// TIA Portal V20 export
VAR_GLOBAL   // PLC tag table "Default tag table"
   SAFETY_TEST AT %M200.0 : Bool;
   Tag_1 AT %M200.1 : Bool;
   Tag_3 AT %M2000.0 : Bool;
   Tag_4 AT %M2000.1 : Bool;
   armsMainValve AT %Q1557.0 : Bool;
   clampsMainValve AT %Q1557.1 : Bool;
   Tag_5 AT %M2001.0 : Bool;
   Tag_6 AT %M2001.1 : Bool;
   Tag_7 AT %M2001.3 : Bool;
   Tag_8 AT %M2001.2 : Bool;
   Tag_9 AT %M222.2 : Bool;
   SS2_R1_STO AT %Q150.0 : Bool;
   Tag_11 AT %M222.3 : Bool;
   Tag_10 AT %M212.0 : Bool;
   Tag_12 AT %M500.0 : Bool;
   Tag_13 AT %M500.1 : Bool;
   Tag_14 AT %M500.2 : Bool;
   Tag_15 AT %M501.0 : Bool;
   Tag_16 AT %M501.1 : Bool;
   TipHydContactorFB AT %I2105.0 : Bool;
   S2_R2_STO AT %Q169.0 : Bool;
   Tag_17 AT %M3000.0 : Bool;
   Tag_18 AT %M3000.1 : Bool;
   Tag_2 AT %M222.4 : Bool;
   Tag_19 AT %M222.5 : Bool;
   CS_Drive_PL_Actor_Interface_AddressIn AT %I50.0 : "PD_TEL105_IN";
   CS_Drive_PP_Actor_Interface_AddressIn AT %I18.0 : "PD_TEL105_IN";
   CS_Drive_TL_Actor_Interface_AddressIn AT %I102.0 : "PD_TEL105_IN";
   CS_Drive_TP_Actor_Interface_AddressIn AT %I76.0 : "PD_TEL105_IN";
   "CS_Drive_PL_Actor_Interface_AddressIn(1)" AT %I50.0 : "PD_TEL1_IN";
   CS_Drive_PL_Actor_Interface_AddressOut AT %Q50.0 : "PD_TEL105_OUT";
   CS_Drive_PP_Actor_Interface_AddressOut AT %Q18.0 : "PD_TEL105_OUT";
   CS_Drive_TL_Actor_Interface_AddressOut AT %Q102.0 : "PD_TEL105_OUT";
   CS_Drive_TP_Actor_Interface_AddressOut AT %Q76.0 : "PD_TEL105_OUT";
   "CS_Drive_PL_Actor_Interface_AddressOut(1)" AT %Q50.0 : "PD_TEL1_OUT";
   Clock_Byte AT %MB1000 : Byte;
   Clock_10Hz AT %M1000.0 : Bool;
   Clock_5Hz AT %M1000.1 : Bool;
   "Clock_2.5Hz" AT %M1000.2 : Bool;
   Clock_2Hz AT %M1000.3 : Bool;
   "Clock_1.25Hz" AT %M1000.4 : Bool;
   Clock_1Hz AT %M1000.5 : Bool;
   "Clock_0.625Hz" AT %M1000.6 : Bool;
   "Clock_0.5Hz" AT %M1000.7 : Bool;
   Tag_20 AT %M600.0 : Bool;
   Tag_22 AT %Q600.3 : Bool;
   SS1_R1_STO AT %Q122.0 : Bool;
   SS1_R1_ACK_STO AT %Q122.7 : Bool;
   SS1_R2_STO AT %Q131.0 : Bool;
   SS1_R2_ACK_STO AT %Q131.7 : Bool;
   Tag_23 AT %Q400.3 : Bool;
   Tag_24 AT %M666.0 : Bool;
   "SS1_R1_STO(1)" AT %Q896.0 : Bool;
   "SS1_R2_STO(1)" AT %Q915.0 : Bool;
   Tag_21 AT %M2222.0 : Bool;
   SpeedAxis_1_Actor_Interface_AddressIn AT %I345.0 : "PD_TEL1_IN";
   SpeedAxis_1_Actor_Interface_AddressOut AT %Q344.0 : "PD_TEL1_OUT";
   Tag_25 AT %M999.0 : Bool;
   Tag_26 AT %M999.1 : Bool;
   Tag_27 AT %M999.2 : Bool;
   "CS_Drive_PL_Actor_Interface_AddressIn(3)" AT %I120.0 : "PD_TEL105_IN";
   "CS_Drive_PL_Actor_Interface_AddressOut(3)" AT %Q120.0 : "PD_TEL105_OUT";
   "CS_Drive_PL_Actor_Interface_AddressIn(4)" AT %I1157.0 : "PD_TEL3_IN";
   "CS_Drive_PL_Actor_Interface_AddressOut(4)" AT %Q1157.0 : "PD_TEL3_OUT";
   Tag_28 AT %Q1175.0 : Bool;
   Tag_29 AT %Q1175.1 : Bool;
   Tag_30 AT %M444.0 : Bool;
   "CS_Drive_PP_Actor_Interface_AddressIn(1)" AT %I120.0 : "PD_TEL3_IN";
   "CS_Drive_PP_Actor_Interface_AddressOut(1)" AT %Q0.0 : "PD_TEL3_OUT";
   STO_CS_PL AT %Q393.0 : Bool;
   "CS_Drive_PL_Actor_Interface_AddressIn(5)" AT %I1177.0 : "PD_TEL105_IN";
   "CS_Drive_PL_Actor_Interface_AddressOut(5)" AT %Q1177.0 : "PD_TEL105_OUT";
   "CS_Drive_PP_Actor_Interface_AddressIn(2)" AT %I1157.0 : "PD_TEL105_IN";
   "CS_Drive_PP_Actor_Interface_AddressOut(2)" AT %Q1157.0 : "PD_TEL105_OUT";
   "CS_Drive_TL_Actor_Interface_AddressIn(1)" AT %I1203.0 : "PD_TEL105_IN";
   "CS_Drive_TL_Actor_Interface_AddressOut(1)" AT %Q1203.0 : "PD_TEL105_OUT";
   "CS_Drive_TP_Actor_Interface_AddressIn(1)" AT %I1223.0 : "PD_TEL105_IN";
   "CS_Drive_TP_Actor_Interface_AddressOut(1)" AT %Q1223.0 : "PD_TEL105_OUT";
   STO_CS_PP AT %Q643.0 : Bool;
   STO_CS_TP AT %Q1140.0 : Bool;
   STO_CS_TL AT %Q1243.0 : Bool;
   Tag_33 AT %M777.0 : Bool;
   Tag_34 AT %M777.1 : Bool;
   Tag_35 AT %M777.3 : Bool;
   Tag_36 AT %M777.5 : Bool;
   Tag_37 AT %M777.6 : Bool;
   Tag_38 AT %M777.7 : Bool;
   Tag_39 AT %M778.1 : Bool;
   Tag_40 AT %M888.0 : Bool;
   Tag_41 AT %M779.0 : Bool;
   CS_QR_Reader AT %IW5002 : Word;
   QR_Reader AT %ID5000 : DWord;
   Tag_43 AT %M832.0 : Bool;
   STO_CS_R1 AT %Q226.0 : Bool;
   STO_CS_R2 AT %Q245.0 : Bool;
   Tag_31 AT %IW5000 : Word;
   STO_CSM1 AT %Q188.0 : Bool;
   STO_CSM2 AT %Q207.0 : Bool;
   Tag_32 AT %M657.4 : Bool;
   CC_Vibrating_Unit_1_Actor_Interface_AddressIn AT %I446.0 : "PD_TEL1_IN";
   CC_Vibrating_Unit_1_Actor_Interface_AddressOut AT %Q445.0 : "PD_TEL1_OUT";
   CC_Vibrating_Unit_3_Actor_Interface_AddressIn AT %I544.0 : "PD_TEL1_IN";
   CC_Vibrating_Unit_3_Actor_Interface_AddressOut AT %Q544.0 : "PD_TEL1_OUT";
   CC_Vibrating_Unit_2_Actor_Interface_AddressIn AT %I495.0 : "PD_TEL1_IN";
   CC_Vibrating_Unit_2_Actor_Interface_AddressOut AT %Q494.0 : "PD_TEL1_OUT";
   Tag_42 AT %M946.0 : Bool;
   Tag_44 AT %MB856 : Byte;
   STO_MST30B AT %Q1115.0 : Bool;
   STO_MST29 AT %Q1257.0 : Bool;
   Tag_45 AT %M442.0 : Bool;
   Tag_46 AT %M445.0 : Bool;
   Tag_47 AT %M558.4 : Bool;
   Tag_48 AT %M487.4 : Bool;
   Tag_49 AT %M699.1 : Bool;
   Tag_50 AT %M467.0 : Bool;
   Tag_51 AT %M788.5 : Bool;
   Tag_52 AT %M376.4 : Bool;
   Tag_53 AT %M35.4 : Bool;
   Tag_54 AT %M323.3 : Bool;
   Tag_55 AT %M452.3 : Bool;
   Tag_56 AT %M669.3 : Bool;
   Tag_57 AT %M100.3 : Bool;
   Tag_58 AT %Q2250.1 : Bool;
   Tag_59 AT %M836.4 : Bool;
   Tag_60 AT %M816.0 : Bool;
   Tag_61 AT %M997.0 : Bool;
   Tag_62 AT %M100.0 : Bool;
   Tag_63 AT %M899.6 : Bool;
   CS_Drive_PL_Actor_Interface_TorqueDataAddressIn AT %I1294.0 : "PD_TEL750_IN";
   CS_Drive_PL_Actor_Interface_TorqueDataAddressOut AT %Q1294.0 : "PD_TEL750_OUT";
   CS_Drive_PP_Actor_Interface_TorqueDataAddressIn AT %I1420.0 : "PD_TEL750_IN";
   CS_Drive_PP_Actor_Interface_TorqueDataAddressOut AT %Q1420.0 : "PD_TEL750_OUT";
   CS_Drive_TL_Actor_Interface_TorqueDataAddressIn AT %I1426.0 : "PD_TEL750_IN";
   CS_Drive_TL_Actor_Interface_TorqueDataAddressOut AT %Q1426.0 : "PD_TEL750_OUT";
   CS_Drive_TP_Actor_Interface_TorqueDataAddressIn AT %I1432.0 : "PD_TEL750_IN";
   CS_Drive_TP_Actor_Interface_TorqueDataAddressOut AT %Q1432.0 : "PD_TEL750_OUT";
   Tag_64 AT %M655.3 : Bool;
   Tag_65 AT %M599.1 : Bool;
   Tag_66 AT %M476.2 : Bool;
   Tag_67 AT %M888.2 : Bool;
   Tag_68 AT %M444.3 : Bool;
   Tag_69 AT %M398.4 : Bool;
   Tag_70 AT %M1333.0 : Bool;
   Tag_71 AT %M611.2 : Bool;
   Tag_72 AT %M611.3 : Bool;
   Tag_73 AT %M833.4 : Bool;
   Tag_74 AT %M881.1 : Bool;
   Tag_75 AT %M71.0 : Bool;
   Tag_76 AT %M727.1 : Bool;
END_VAR
